// LS Electric XG5000 project: 통테
// PLC LSPLC

PROGRAM NewProgram (task: 스캔 프로그램)

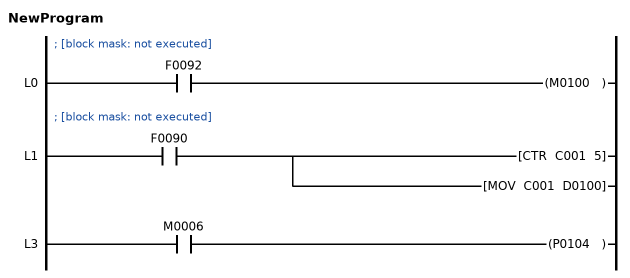
; L0 (block mask: not executed)
LOAD      F0092
OUT       M0100
; L1 (block mask: not executed)
LOAD      F0090
CTR       C001 5
MOV       C001 D0100
; L3
LOAD      M0006
OUT       P0104